Yaskawa INFORM job: X2_DOD_HARDOX_1(90,180).JBI

/JOB
//NAME X2_DOD_HARDOX_1(90,180)
//POS
///NPOS 279,279,279,21,0,0
///TOOL 0
///POSTYPE PULSE
///PULSE
C00000=3109,-122452,-100913,-73,83322,449
C00001=-118807,-122452,-100913,-73,83322,449
C00002=-118807,-122452,-100913,-73,83322,449
C00003=-118807,-122452,-100911,-58,83321,449
C00004=-118807,-121735,-99413,-58,82766,449
C00005=-118807,-121842,-99633,-58,82848,449
C00006=-118839,-119744,-98985,-56,83526,438
C00007=-118804,-122923,-101491,-58,83435,450
C00008=-97639,-115747,-96446,15703,79249,7339
C00009=-97639,-115388,-95597,15719,78924,7296
C00010=-97639,-114939,-94559,15740,78531,7244
C00011=-97639,-115025,-94759,15735,78607,7253
C00012=-98061,-112826,-94039,15753,79350,7198
C00013=-97812,-116320,-99930,15652,81066,7508
C00014=-101587,-63576,-81599,5795,100855,28886
C00015=-101047,-68280,-81443,-762,96025,52675
C00016=-101825,-68101,-80196,-684,95342,52421
C00017=-101825,-68359,-78475,-683,94153,52425
C00018=-101825,-68340,-78625,-683,94255,52425
C00019=-102365,-71446,-80148,-632,93594,52249
C00020=-101826,-68339,-78622,-682,94255,52423
C00021=-102743,-68014,-78460,-592,94316,52120
C00022=-104230,-67130,-78018,-446,94488,51627
C00023=-101826,-68180,-79726,-683,95016,52419
C00024=-105406,-85017,-88644,8711,87087,51760
C00025=-104819,-84637,-86896,8622,86156,51894
C00026=-104819,-84584,-85262,8627,85189,51829
C00027=-104821,-84590,-85434,8628,85291,51834
C00028=-104466,-81413,-84026,8564,86011,52005
C00029=-122297,-70560,-77685,25207,96114,48988
C00030=-122297,-70602,-76512,25163,95437,48844
C00031=-120462,-72211,-77291,25034,94575,49337
C00032=-120807,-72109,-79837,25145,96151,49547
C00033=-93546,-62658,-75100,22039,90269,58200
C00034=-94184,-63290,-73954,22130,89476,57830
C00035=-94067,-63307,-72915,22106,88843,57754
C00036=-94003,-63340,-73099,22003,88907,57787
C00037=-94409,-63618,-73243,22068,88963,57653
C00038=-94117,-63207,-75013,22033,90096,57964
C00039=-99361,-30382,-55480,23023,95964,57224
C00040=-99566,-28855,-54147,23052,95988,57159
C00041=-99566,-29275,-52787,22997,95015,56970
C00042=-99566,-29231,-52941,23002,95123,56991
C00043=-99913,-29435,-53082,23054,95198,56882
C00044=-99765,-28813,-54689,23103,96366,57161
C00045=-70126,-14814,-46677,22990,86577,66649
C00046=-69225,-6747,-37988,28306,84286,67688
C00047=-68210,-7965,-38259,28007,83556,67874
C00048=-68210,-8415,-36953,28052,82637,67651
C00049=-68211,-8369,-37103,28046,82745,67677
C00050=-67132,-7971,-36789,27709,82413,67989
C00051=-68211,-8369,-37103,28046,82745,67677
C00052=-69273,3622,-28812,29896,91299,69888
C00053=-69171,1587,-30541,29875,91281,69920
C00054=-67356,-7788,-38801,27721,83669,68208
C00055=-69304,23814,-19677,20373,105408,54389
C00056=-63772,25809,-17813,13128,104960,54938
C00057=-63772,25417,-17229,13089,104414,54876
C00058=-63772,25480,-17328,13095,104505,54886
C00059=-64757,25100,-17697,13206,104683,54580
C00060=-63772,25480,-17328,13095,104505,54886
C00061=-68307,7319,-30798,19970,94187,53100
C00062=-68472,9999,-28438,20005,94151,53039
C00063=-64638,26032,-18396,13259,105551,54716
C00064=-73474,52417,-1620,14466,110043,52326
C00065=-77083,27840,-18357,21376,94830,50068
C00066=-77083,27429,-17836,21353,94333,49979
C00067=-77083,27542,-17981,21360,94470,50004
C00068=-77263,29809,-15685,21397,94280,49912
C00069=-77083,27542,-17981,21360,94470,50004
C00070=-83249,15329,-22913,33380,85893,48144
C00071=-82325,15284,-22953,33088,85562,48389
C00072=-77119,30179,-17426,21415,95423,50164
C00073=-76952,50122,-2257,13631,106723,63183
C00074=-76686,48992,-1778,13529,105834,63166
C00075=-76686,48070,-780,13449,104775,63046
C00076=-76686,48153,-875,13455,104873,63057
C00077=-76611,45681,-3555,13472,105231,63123
C00078=-76686,48153,-875,13455,104873,63057
C00079=-77765,47797,-1260,13598,105089,62727
C00080=-77503,48179,-2005,13615,105687,62882
C00081=-102232,64721,13378,16026,108849,55032
C00082=-108949,82207,34418,16047,106253,52367
C00083=-109653,82825,36624,15990,105380,52004
C00084=-109653,82216,37670,15908,104457,51880
C00085=-109653,82279,37553,15917,104559,51893
C00086=-109965,79801,34505,15982,105197,51872
C00087=-109653,82279,37553,15917,104559,51893
C00088=-109989,64914,17803,16949,99513,51403
C00089=-109412,64226,17005,16864,99534,51598
C00090=-110036,80923,34280,16050,105899,51944
C00091=-104345,57087,4731,-4349,89209,83366
C00092=-104496,43008,-4738,-4784,85361,83353
C00093=-104479,42314,-3820,-4795,84443,83394
C00094=-104496,42365,-3916,-4789,84527,83385
C00095=-104255,44770,-1355,-4879,84201,83473
C00096=-104496,42365,-3916,-4789,84527,83385
C00097=-105699,43472,-2745,-4351,84311,83020
C00098=-104155,44462,-3948,-4908,85640,83449
C00099=-104173,44480,-3904,-4901,85622,83444
C00100=-106809,29779,-23791,-3960,104541,82225
C00101=-101987,32580,-18779,-13564,104520,81725
C00102=-101987,31981,-18214,-13517,103880,81798
C00103=-101987,32158,-18384,-13531,104070,81776
C00104=-101545,36557,-13887,-13574,103641,81966
C00105=-101545,36395,-13728,-13561,103461,81987
C00106=-101706,33738,-16315,-13551,103657,81914
C00107=-101764,35134,-16470,-13596,104438,81806
C00108=-104548,23177,-32201,15979,107404,88348
C00109=-105455,19857,-30331,15882,104803,87705
C00110=-105493,19341,-29883,15843,104288,87624
C00111=-105493,19514,-30048,15860,104471,87649
C00112=-105050,22772,-26945,15761,104169,87752
C00113=-105050,22547,-26726,15741,103926,87719
C00114=-105181,21576,-27656,15770,104020,87688
C00115=-105214,23260,-28464,15890,105337,87854
C00116=-132284,21592,-30078,20050,110667,79822
C00117=-127713,47562,-3500,19091,106863,80708
C00118=-127298,48428,-1312,18938,105922,80691
C00119=-127298,47930,-750,18875,105351,80598
C00120=-127298,48117,-965,18899,105568,80634
C00121=-126552,50894,2078,18759,104988,80792
C00122=-126552,50661,2355,18730,104712,80748
C00123=-126852,49777,1385,18779,104913,80679
C00124=-126833,51121,1366,18850,105576,80792
C00125=-130599,55255,6018,19225,105667,79530
C00126=-130503,55108,6106,19201,105525,79539
C00127=-130503,54617,6701,19135,104939,79443
C00128=-130503,54765,6517,19154,105119,79472
C00129=-129703,58202,10396,18998,104360,79621
C00130=-129703,58014,10641,18975,104124,79585
C00131=-129980,56421,8841,19034,104460,79543
C00132=-129931,58896,8732,19166,105718,79766
C00133=-131687,18895,-22844,22845,77130,75091
C00134=-123291,20715,-19983,19085,74393,77453
C00135=-123291,20226,-19115,19152,73648,77333
C00136=-123291,20408,-19449,19125,73931,77379
C00137=-123978,17743,-21949,19433,74239,77195
C00138=-123978,17498,-21504,19467,73861,77134
C00139=-123624,18839,-20254,19309,73708,77231
C00140=-123896,19533,-21399,19345,74771,77313
C00141=-129275,29738,-11535,21888,75238,75561
C00142=-129239,30151,-9876,21947,74475,75432
C00143=-129239,29906,-9384,21989,74076,75357
C00144=-129239,29966,-9509,21979,74176,75376
C00145=-128682,29827,-9665,21723,74091,75555
C00146=-129188,29970,-9523,21952,74204,75400
C00147=-129412,25077,-15126,21963,75128,75497
C00148=-127801,23871,-15548,21269,74401,75919
C00149=-127478,25278,-14188,21132,74217,75998
C00150=-127515,25076,-16775,21017,75619,76237
C00151=-133346,41405,-239,23776,75434,74185
C00152=-133209,40965,432,23780,74810,74105
C00153=-133209,40606,1199,23846,74209,73980
C00154=-133209,40709,971,23826,74386,74016
C00155=-134183,37129,-2750,24201,75064,73812
C00156=-134183,36974,-2419,24229,74805,73759
C00157=-133761,38534,-808,24066,74516,73849
C00158=-133829,37887,-2909,24000,75417,74012
C00159=-156022,88654,55414,33609,74162,65271
C00160=-155367,67510,26868,18073,74568,63363
C00161=-155657,68026,27393,18196,74574,63263
C00162=-155657,67713,28231,18251,73929,63165
C00163=-155657,67848,27854,18227,74216,63209
C00164=-157091,64685,24164,18764,75139,62855
C00165=-157091,64518,24594,18793,74808,62803
C00166=-156451,66014,26335,18558,74384,62959
C00167=-156599,65406,24098,18535,75428,63070
C00168=-129275,29738,-11535,21888,75238,75561
C00169=-129021,46521,3990,22011,82280,76800
C00170=-127853,72870,28739,19070,95872,81441
C00171=-127868,72875,28745,19073,95874,81436
C00172=-128195,57479,12526,19645,90783,80632
C00173=-130174,39740,-1969,24825,82186,79427
C00174=-129425,38207,-3565,24549,82155,79680
C00175=-125055,30126,-11758,22903,81812,81108
C00176=-125820,29533,-14095,23141,83054,81090
C00177=-116935,30569,-15261,-2620,77337,75322
C00178=-116946,32606,-9583,-2640,74890,75373
C00179=-117027,32230,-9962,-2601,74928,75346
C00180=-117027,32230,-9962,-2601,74928,75346
C00181=-116186,24046,-15173,-4825,69577,75450
C00182=-116977,23560,-15650,-4179,69663,75252
C00183=-117705,24065,-15165,-3796,69592,75013
C00184=-121349,29184,-10162,-1867,69024,73811
C00185=-155953,64784,27397,14502,67420,61519
C00186=-160308,74014,38140,24557,70405,61761
C00187=-162428,80563,46699,30040,71499,61878
C00188=-162835,78141,41049,29865,73587,62284
C00189=-131165,66178,18557,19074,103796,79028
C00190=-132263,70632,26138,21339,107315,79548
C00191=-130805,66688,21488,21399,107742,80153
C00192=-126998,57798,11204,21464,108466,81651
C00193=-126971,60939,9833,21835,110752,82102
C00194=-128691,16256,-41784,23758,119313,83319
C00195=-126023,-4907,-54781,25051,118959,68774
C00196=-124897,-8515,-53636,24373,116335,68560
C00197=-119086,-23897,-66107,13265,108526,66827
C00198=-120519,-17402,-59352,23947,114251,69687
C00199=-120519,-17402,-59352,23947,114251,69687
C00200=-122564,-44453,-75136,25957,97391,66445
C00201=-123228,-71474,-85542,26631,77979,61978
C00202=-105873,-76739,-89965,2224,72297,65038
C00203=-111330,-72335,-87900,4522,73506,63229
C00204=-111330,-72335,-87900,4522,73506,63229
C00205=-112163,-45580,-78612,3641,93445,63594
C00206=-119086,-23897,-66107,13265,108526,66827
C00207=-125757,-8552,-54820,24574,117205,68447
C00208=-88641,48412,-4226,20715,106428,79236
C00209=-87799,48144,-1656,20397,104625,79199
C00210=-87620,46255,-1934,20290,103831,79122
C00211=-86307,38945,-9666,20202,104482,79674
C00212=-86372,39978,-10015,20293,105198,79777
C00213=-77383,-1492,-44705,4977,83394,77592
C00214=-77548,-1237,-43087,5052,82544,77506
C00215=-83219,23182,-25333,15019,98405,78867
C00216=-80942,13133,-33032,25463,110902,83847
C00217=-81045,14451,-33580,25670,111852,84035
C00218=-73165,-12601,-57571,12637,98383,82001
C00219=-73127,-13258,-56291,12584,97280,81900
C00220=-74782,-8289,-52590,17954,103500,83219
C00221=-74719,-7609,-53088,18001,104113,83334
C00222=-82838,36617,-17283,19543,106393,81060
C00223=-68187,-8044,-38286,28001,83527,67876
C00224=-68187,-8044,-38286,28001,83527,67876
C00225=-67058,-9477,-38022,27689,82372,68007
C00226=-68116,3817,-27265,27987,82912,67789
C00227=-68116,3817,-27265,27987,82912,67789
C00228=-64919,-4904,-34321,21162,76650,66545
C00229=-61528,17256,-21731,13706,92976,69906
C00230=-58415,32145,-10038,7508,102141,70514
C00231=-57465,27559,-14703,8015,104960,71103
C00232=-57465,27559,-14703,8015,104960,71103
C00233=-65198,47488,8134,19223,111073,70945
C00234=-67034,-9554,-38047,27682,82343,68009
C00235=-67251,-9396,-39953,27695,83527,68213
C00236=-83600,19181,-26002,32561,94222,65167
C00237=-77066,27753,-18406,21371,94813,50070
C00238=-76689,29778,-15601,21234,94082,50062
C00239=-76186,35433,-13032,12668,99412,49208
C00240=-76186,35433,-13032,12668,99412,49208
C00241=-74826,30522,-18009,8636,97794,54751
C00242=-79416,42076,-6372,17402,103035,66342
C00243=-86419,39929,-2219,28404,103150,66219
C00244=-84052,39875,-2276,28113,102413,66901
C00245=-84052,39875,-2276,28113,102413,66901
C00246=-81568,19785,-21142,23805,91116,64901
C00247=-82431,9786,-27697,23195,82999,70057
C00248=-82776,9522,-31565,23250,85160,70361
C00249=-89191,6029,-42138,6806,101823,66252
C00250=-95828,93776,43903,513,93919,62536
C00251=-104499,43028,-4714,-4783,85356,83352
C00252=-108433,63055,13709,2825,95010,83470
C00253=-107826,61367,13148,420,94873,83225
C00254=-107008,65665,17554,6129,98722,84709
C00255=-107008,65665,17554,6129,98722,84709
C00256=-106682,56060,7916,7154,93832,84823
C00257=-104948,47222,-158,3217,88060,84363
C00258=-103642,41840,-4077,-3525,83464,83442
C00259=-105882,43444,-2375,-2683,83163,82753
C00260=-105882,43444,-2375,-2683,83163,82753
C00261=-104950,42848,-3229,-5574,83910,82481
C00262=-107826,61367,13148,420,94873,83225
C00263=-106192,65684,14431,-2737,97774,82157
C00264=-82945,4708,-44686,-381,111426,77490
C00265=-79819,-2415,-47658,-697,109614,78498
C00266=-78726,-4935,-47947,-802,108508,78855
C00267=-78978,-4815,-47850,-776,108508,78773
C00268=-82498,-4521,-47863,-435,108644,77640
C00269=-91525,7946,-35181,-15697,111008,71310
C00270=-91286,10128,-36695,-15968,113029,71106
C00271=-98325,-60487,-84418,-569,84750,74718
C00272=-131349,-72907,-81893,29779,75628,65053
C00273=-129293,-70616,-79214,29166,74512,65558
C00274=-88918,-58369,-72899,11987,66692,79059
C00275=-87177,-56818,-72056,11108,66724,79688
C00276=-87910,-58429,-75945,11347,68359,79585
C00277=-85222,-130765,-111241,11638,52830,79008
C00278=3322,-122452,-100913,-73,83322,449
BC00000=198923,666220,911653
BC00001=316579,666220,219283
BC00002=307984,758478,148723
BC00003=307985,760782,131305
BC00004=307985,760782,131305
BC00005=307985,760782,131305
BC00006=307985,760782,131305
BC00007=307985,760782,131305
BC00008=307985,760782,131305
BC00009=307985,760782,131305
BC00010=307985,760782,131305
BC00011=307985,760782,131305
BC00012=307985,760782,131305
BC00013=307985,760782,131305
BC00014=307985,760782,131305
BC00015=307985,760782,131305
BC00016=307985,760782,131305
BC00017=307985,760782,131305
BC00018=307985,760782,131305
BC00019=307985,760782,131305
BC00020=307985,760782,131305
BC00021=307985,760782,131305
BC00022=307985,760782,131305
BC00023=307985,760782,131305
BC00024=307985,760782,131305
BC00025=307985,760782,131305
BC00026=307985,760782,131305
BC00027=307985,760782,131305
BC00028=307985,760782,131305
BC00029=307985,760782,131305
BC00030=307985,760782,131305
BC00031=307985,760782,131305
BC00032=307985,760782,131305
BC00033=307986,760782,131302
BC00034=307986,760782,131302
BC00035=307986,760782,131302
BC00036=307986,760782,131302
BC00037=307986,760782,131302
BC00038=307986,760782,131302
BC00039=307986,760782,131302
BC00040=307986,760782,131302
BC00041=307986,760782,131302
BC00042=307986,760782,131302
BC00043=307986,760782,131302
BC00044=307986,760782,131302
BC00045=258907,777593,97712
BC00046=258907,777593,97712
BC00047=258907,777593,97712
BC00048=258907,777593,97712
BC00049=258907,777592,97711
BC00050=258907,777592,97711
BC00051=258907,777592,97711
BC00052=258907,777592,97711
BC00053=258907,777592,97711
BC00054=258907,777592,97711
BC00055=274910,772479,88149
BC00056=274910,772479,88149
BC00057=274910,772479,88149
BC00058=274910,772479,88149
BC00059=274910,772479,88149
BC00060=274910,772479,88149
BC00061=274910,772479,88149
BC00062=274910,772479,88149
BC00063=274910,772479,88149
BC00064=280793,772479,47450
BC00065=280793,772479,47450
BC00066=280793,772479,47450
BC00067=280793,772479,47450
BC00068=280793,772479,47450
BC00069=280793,772479,47450
BC00070=280793,772479,47450
BC00071=280793,772479,47450
BC00072=280793,772479,47450
BC00073=280793,772479,47450
BC00074=280793,772479,47450
BC00075=280793,772479,47450
BC00076=280793,772479,47450
BC00077=280793,772479,47450
BC00078=280793,772479,47450
BC00079=280793,772479,47450
BC00080=280793,772479,47450
BC00081=311515,772478,37762
BC00082=328438,772478,37762
BC00083=328438,772478,37762
BC00084=328438,772478,37762
BC00085=328438,772478,37762
BC00086=328438,772478,37762
BC00087=328438,772478,37762
BC00088=328438,772478,37762
BC00089=328438,772478,37762
BC00090=328438,772478,37762
BC00091=328438,772478,37762
BC00092=328438,772478,37762
BC00093=328438,772478,37762
BC00094=328438,772478,37762
BC00095=328438,772478,37762
BC00096=328438,772478,37762
BC00097=328438,772478,37762
BC00098=328438,772478,37762
BC00099=308564,725534,37762
BC00100=308564,725534,37762
BC00101=308564,725534,37762
BC00102=308564,725534,37762
BC00103=308564,725534,37762
BC00104=308564,725534,37762
BC00105=308564,725534,37762
BC00106=308564,725534,37762
BC00107=308564,725534,37762
BC00108=308564,725534,37762
BC00109=308564,725534,37762
BC00110=308564,725534,37762
BC00111=308564,725534,37762
BC00112=308564,725534,37762
BC00113=308564,725534,37762
BC00114=308564,725534,37762
BC00115=308564,725534,37762
BC00116=308564,725534,37762
BC00117=308564,725534,37762
BC00118=308564,725534,37762
BC00119=308564,725534,37762
BC00120=308564,725534,37762
BC00121=308564,725534,37762
BC00122=308564,725534,37762
BC00123=308564,725534,37762
BC00124=308564,725534,37762
BC00125=308564,725534,37762
BC00126=308564,725534,37762
BC00127=308564,725534,37762
BC00128=308564,725534,37762
BC00129=308564,725534,37762
BC00130=308564,725534,37762
BC00131=308564,725534,37762
BC00132=308564,725534,37762
BC00133=308564,725534,37762
BC00134=308564,725534,37762
BC00135=308564,725534,37762
BC00136=308564,725534,37762
BC00137=308564,725534,37762
BC00138=308564,725534,37762
BC00139=308564,725534,37762
BC00140=308564,725534,37762
BC00141=308564,725534,37762
BC00142=308564,725534,37762
BC00143=308564,725534,37762
BC00144=308564,725534,37762
BC00145=308564,725534,37762
BC00146=308564,725534,37762
BC00147=308564,725534,37762
BC00148=308564,725534,37762
BC00149=308564,725534,37762
BC00150=308564,725534,37762
BC00151=308564,725534,37761
BC00152=308564,725534,37761
BC00153=308564,725534,37761
BC00154=308564,725534,37761
BC00155=308564,725534,37761
BC00156=308564,725534,37761
BC00157=308564,725534,37761
BC00158=308564,725534,37761
BC00159=362000,725534,37761
BC00160=362000,752970,37761
BC00161=362000,752970,37761
BC00162=362000,752970,37761
BC00163=362000,752970,37761
BC00164=362000,752970,37761
BC00165=362000,752970,37761
BC00166=362000,752970,37761
BC00167=362000,752970,37761
BC00168=308564,725534,37762
BC00169=308564,725534,37762
BC00170=308564,725534,37762
BC00171=308564,725534,37762
BC00172=308564,725534,37762
BC00173=308564,725534,37762
BC00174=308564,725534,37762
BC00175=308564,725534,37762
BC00176=308564,725534,37762
BC00177=308564,725534,37762
BC00178=308564,725534,37762
BC00179=308564,725534,37762
BC00180=308564,725534,37762
BC00181=308564,725534,37762
BC00182=308564,725534,37762
BC00183=308564,725534,37762
BC00184=308564,725534,37762
BC00185=362000,752970,37761
BC00186=362000,752970,37761
BC00187=362000,752970,37761
BC00188=362000,752970,37761
BC00189=308564,725534,37762
BC00190=308564,725534,37762
BC00191=308564,725534,37762
BC00192=308564,725534,37762
BC00193=308564,725534,37762
BC00194=308564,725534,37762
BC00195=308564,725534,37762
BC00196=308564,725534,37762
BC00197=308564,725534,37762
BC00198=308564,725534,37762
BC00199=308564,725534,37762
BC00200=308564,725534,37762
BC00201=308564,725534,37762
BC00202=308564,725534,37762
BC00203=308564,725534,37762
BC00204=308564,725534,37762
BC00205=308564,725534,37762
BC00206=308564,725534,37762
BC00207=308564,725534,37762
BC00208=255253,725534,37762
BC00209=255253,725534,37762
BC00210=255253,725534,37762
BC00211=255253,725534,37762
BC00212=255253,725534,37762
BC00213=255253,725534,37762
BC00214=255254,725534,37762
BC00215=255253,725534,37762
BC00216=255253,725534,37762
BC00217=255253,725534,37762
BC00218=255253,725534,37762
BC00219=255253,725534,37762
BC00220=255253,725534,37762
BC00221=255253,725534,37762
BC00222=255253,725534,37762
BC00223=258907,777593,97712
BC00224=258907,777593,97712
BC00225=258907,777593,97712
BC00226=259033,777461,97560
BC00227=259033,777461,97560
BC00228=259039,777455,97553
BC00229=259039,777455,97553
BC00230=259100,772345,97480
BC00231=259100,773616,97479
BC00232=259100,773616,97479
BC00233=261144,764069,97479
BC00234=258907,777593,97712
BC00235=258907,777593,97712
BC00236=281642,777593,57012
BC00237=280793,772479,47450
BC00238=280794,772478,47449
BC00239=280809,772452,47444
BC00240=280809,772452,47444
BC00241=280809,772452,47444
BC00242=280808,772453,47444
BC00243=293831,772390,68911
BC00244=293831,772390,68911
BC00245=293831,772390,68911
BC00246=293831,772390,68911
BC00247=293831,772390,68911
BC00248=293831,772390,68911
BC00249=293831,772390,68911
BC00250=293831,746596,7862
BC00251=328438,772478,37762
BC00252=328438,772478,37762
BC00253=328438,772478,37762
BC00254=328370,772478,37776
BC00255=328370,772478,37776
BC00256=328370,772478,37776
BC00257=328370,772478,37776
BC00258=328280,772478,37857
BC00259=328280,772478,37857
BC00260=328280,772478,37857
BC00261=328280,772478,37857
BC00262=328438,772478,37762
BC00263=328280,772478,37857
BC00264=293831,772391,68907
BC00265=293831,772391,68906
BC00266=293831,772391,68906
BC00267=293831,772391,68906
BC00268=293831,772391,68906
BC00269=293831,772391,68906
BC00270=293831,772391,68906
BC00271=274540,694640,68906
BC00272=274540,694640,68906
BC00273=274540,694640,68906
BC00274=274540,694640,68906
BC00275=274540,694640,68906
BC00276=274540,694640,68906
BC00277=274540,694640,68906
BC00278=87761,666220,1075229
EC00000=798156,1112951
EC00001=798156,1112951
EC00002=798156,1112951
EC00003=798155,1112950
EC00004=798155,1112950
EC00005=798155,1112950
EC00006=798155,1112950
EC00007=798155,1112950
EC00008=798155,1112950
EC00009=798155,1112950
EC00010=798155,1112950
EC00011=798155,1112950
EC00012=798155,1112950
EC00013=798155,1112950
EC00014=798155,1112950
EC00015=798155,1112950
EC00016=798155,1112950
EC00017=798155,1112950
EC00018=798155,1112950
EC00019=798155,1112950
EC00020=798147,1112941
EC00021=798147,1112941
EC00022=798147,1112941
EC00023=798147,1112941
EC00024=798155,1112950
EC00025=798155,1112950
EC00026=798155,1112950
EC00027=798155,1112950
EC00028=798155,1112950
EC00029=798155,1112950
EC00030=798155,1112950
EC00031=798155,1112950
EC00032=798155,1112950
EC00033=798155,1112949
EC00034=798155,1112949
EC00035=798155,1112949
EC00036=798155,1112949
EC00037=798155,1112949
EC00038=798155,1112949
EC00039=798155,1112949
EC00040=798155,1112949
EC00041=798155,1112949
EC00042=798155,1112949
EC00043=798155,1112949
EC00044=798155,1112949
EC00045=798154,1112948
EC00046=798154,1112948
EC00047=798154,1112948
EC00048=798154,1112948
EC00049=798153,1112947
EC00050=798153,1112947
EC00051=798153,1112947
EC00052=798153,1112947
EC00053=798153,1112947
EC00054=798153,1112947
EC00055=798153,1112947
EC00056=798153,1112947
EC00057=798153,1112947
EC00058=798153,1112947
EC00059=798153,1112947
EC00060=798153,1112947
EC00061=798153,1112947
EC00062=798153,1112947
EC00063=798153,1112947
EC00064=798153,1112947
EC00065=798153,1112947
EC00066=798153,1112947
EC00067=798153,1112947
EC00068=798153,1112947
EC00069=798153,1112947
EC00070=798153,1112947
EC00071=798153,1112947
EC00072=798153,1112947
EC00073=798153,1112947
EC00074=798153,1112947
EC00075=798153,1112947
EC00076=798153,1112947
EC00077=798153,1112947
EC00078=798153,1112947
EC00079=798153,1112947
EC00080=798153,1112947
EC00081=798153,1112946
EC00082=798153,1112946
EC00083=798153,1112946
EC00084=798153,1112946
EC00085=798153,1112946
EC00086=798153,1112946
EC00087=798153,1112946
EC00088=798153,1112946
EC00089=798153,1112946
EC00090=798153,1112946
EC00091=798153,1112946
EC00092=798153,1112946
EC00093=798153,1112946
EC00094=798153,1112946
EC00095=798153,1112946
EC00096=798153,1112946
EC00097=798153,1112946
EC00098=798153,1112946
EC00099=798153,1112946
EC00100=798153,1112946
EC00101=798153,1112946
EC00102=798153,1112946
EC00103=798153,1112946
EC00104=798153,1112946
EC00105=798153,1112946
EC00106=798153,1112946
EC00107=798153,1112946
EC00108=798153,1112946
EC00109=798153,1112946
EC00110=798153,1112946
EC00111=798153,1112946
EC00112=798153,1112946
EC00113=798153,1112946
EC00114=798153,1112946
EC00115=798153,1112946
EC00116=798153,1112946
EC00117=798153,1112946
EC00118=798153,1112946
EC00119=798153,1112946
EC00120=798153,1112946
EC00121=798153,1112946
EC00122=798153,1112946
EC00123=798153,1112946
EC00124=798153,1112946
EC00125=798153,1112946
EC00126=798153,1112946
EC00127=798153,1112946
EC00128=798153,1112946
EC00129=798153,1112946
EC00130=798153,1112946
EC00131=798153,1112946
EC00132=798153,1112946
EC00133=798153,1112946
EC00134=798153,1112946
EC00135=798153,1112946
EC00136=798153,1112946
EC00137=798153,1112946
EC00138=798153,1112946
EC00139=798153,1112946
EC00140=798153,1112946
EC00141=798153,1112946
EC00142=798153,1112946
EC00143=798153,1112946
EC00144=798153,1112946
EC00145=798153,1112946
EC00146=798153,1112946
EC00147=798153,1112946
EC00148=798153,1112946
EC00149=798153,1112946
EC00150=798153,1112946
EC00151=798152,1112944
EC00152=798152,1112944
EC00153=798152,1112944
EC00154=798152,1112944
EC00155=798152,1112944
EC00156=798152,1112944
EC00157=798152,1112944
EC00158=798152,1112944
EC00159=798152,1112944
EC00160=798152,1112944
EC00161=798152,1112944
EC00162=798152,1112944
EC00163=798152,1112944
EC00164=798152,1112944
EC00165=798152,1112944
EC00166=798152,1112944
EC00167=798152,1112944
EC00168=798153,1112946
EC00169=798153,1112946
EC00170=798153,1112946
EC00171=798153,1112946
EC00172=798153,1112946
EC00173=798153,1112946
EC00174=798153,1112946
EC00175=798153,1112946
EC00176=798153,1112946
EC00177=798153,1112946
EC00178=798153,1112946
EC00179=798153,1112946
EC00180=798153,1112946
EC00181=798153,1112946
EC00182=798153,1112946
EC00183=798153,1112946
EC00184=798153,1112946
EC00185=798152,1112944
EC00186=798152,1112944
EC00187=798152,1112944
EC00188=798152,1112944
EC00189=798153,1112946
EC00190=798153,1112946
EC00191=798153,1112946
EC00192=798153,1112946
EC00193=798153,1112946
EC00194=798153,1112946
EC00195=798153,1112946
EC00196=798153,1112946
EC00197=798153,1112946
EC00198=798153,1112946
EC00199=798153,1112946
EC00200=798153,1112946
EC00201=798153,1112946
EC00202=798153,1112946
EC00203=798153,1112946
EC00204=798153,1112946
EC00205=798153,1112946
EC00206=798153,1112946
EC00207=798153,1112946
EC00208=798153,1112946
EC00209=798153,1112946
EC00210=798153,1112946
EC00211=798153,1112946
EC00212=798153,1112946
EC00213=798153,1112946
EC00214=798152,1112945
EC00215=798153,1112946
EC00216=798153,1112946
EC00217=798153,1112946
EC00218=798153,1112946
EC00219=798153,1112946
EC00220=798153,1112946
EC00221=798153,1112946
EC00222=798153,1112946
EC00223=798154,1112948
EC00224=798154,1112948
EC00225=798154,1112948
EC00226=798154,1112948
EC00227=798154,1112948
EC00228=798154,1112948
EC00229=798154,1112948
EC00230=798154,1112948
EC00231=798153,1112947
EC00232=798153,1112947
EC00233=798153,1112947
EC00234=798154,1112948
EC00235=798154,1112948
EC00236=798154,1112948
EC00237=798153,1112947
EC00238=798153,1112946
EC00239=798153,1112946
EC00240=798153,1112946
EC00241=798153,1112946
EC00242=798152,1112944
EC00243=798152,1112944
EC00244=798152,1112944
EC00245=798152,1112944
EC00246=798152,1112944
EC00247=798152,1112944
EC00248=798152,1112944
EC00249=798152,1112944
EC00250=798152,1112944
EC00251=798153,1112946
EC00252=798153,1112946
EC00253=798153,1112946
EC00254=798153,1112946
EC00255=798153,1112946
EC00256=798153,1112946
EC00257=798153,1112946
EC00258=798153,1112946
EC00259=798153,1112946
EC00260=798153,1112946
EC00261=798153,1112946
EC00262=798153,1112946
EC00263=798153,1112946
EC00264=798151,1112943
EC00265=798151,1112942
EC00266=798151,1112942
EC00267=798151,1112942
EC00268=798151,1112942
EC00269=798151,1112942
EC00270=798151,1112942
EC00271=798151,1112942
EC00272=798151,1112942
EC00273=798151,1112942
EC00274=798151,1112942
EC00275=798151,1112942
EC00276=798151,1112942
EC00277=798151,1112942
EC00278=798156,1112951
///POSTYPE BASE
///RECTAN
///RCONF 0,0,0,0,0,0,0,0,0,0,0,0,0,0,0,0,0,0,0,0,0,0,0,0
P00006=0.222,-3.123,-1.508,0.0000,0.0000,0.0000
P00021=-0.225,-6.128,-0.405,0.0000,0.0000,0.0000
P00022=0.222,-3.123,-1.508,0.0000,0.0000,0.0000
P00023=0.143,-0.036,0.682,0.0000,0.0000,0.0000
P00024=0.145,-0.552,1.326,0.0000,0.0000,0.0000
P00025=-2.003,0.006,0.728,0.0000,0.0000,0.0000
P00026=0.562,-0.002,-0.337,0.0000,0.0000,0.0000
P00027=-0.746,0.015,-9.096,0.0000,0.0000,0.0000
P00028=-2.237,-0.018,-7.702,0.0000,0.0000,0.0000
P00029=-2.156,-0.086,-4.681,0.0000,0.0000,0.0000
P00030=5.926,-4.294,-1.390,0.0000,0.0000,0.0000
P00031=1.853,-0.001,-1.549,0.0000,0.0000,0.0000
P00032=1.957,0.503,-7.217,0.0000,0.0000,0.0000
///RCONF 0,0,0,0,1,0,0,0,0,0,0,0,0,0,0,0,0,0,0,0,0,0,0,0
P00033=-0.123,0.612,-5.012,0.0000,0.0000,0.0000
///RCONF 0,0,0,0,0,0,0,0,0,0,0,0,0,0,0,0,0,0,0,0,0,0,0,0
P00034=-0.304,0.773,-2.693,0.0000,0.0000,0.0000
P00035=2.817,0.591,-1.622,0.0000,0.0000,0.0000
P00036=-1.108,-0.829,1.850,0.0000,0.0000,0.0000
P00037=0.023,0.937,-2.677,0.0000,0.0000,0.0000
P00038=0.158,-1.133,-1.952,0.0000,0.0000,0.0000
P00039=0.012,-3.081,-0.106,0.0000,0.0000,0.0000
P00040=-0.030,9.648,2.467,0.0000,0.0000,0.0000
//INST
///DATE 2025/03/13 13:01
///ATTR SC,RW
///GROUP1 RB1,BS1
///GROUP2 ST1
NOP
MOVJ C00000 BC00000 VJ=100.00  +MOVJ EC00000 VJ=100.00
MOVJ C00001 BC00001 VJ=100.00  +MOVJ EC00001 VJ=100.00
MOVL C00002 BC00002 V=1000.0  +MOVJ EC00002 VJ=30.00
SFTOF3D
SMOVL C00003 BC00003 V=166.7  +MOVJ EC00003
SREFP 3 C00004 BC00004  +REFP EC00004
CALL JOB:SEARCH-R1-S13D
SET P021 P006
SFTON3D P021
SMOVL C00005 BC00005 V=166.7  +MOVJ EC00005
SREFP 3 C00006 BC00006  +REFP EC00006
CALL JOB:SEARCH-R1-S13D
SET P021 P006
SFTON3D P021
SMOVL C00007 BC00007 V=166.7  +MOVJ EC00007
SFTOF3D
MOVL C00008 BC00008 V=1000.0  +MOVJ EC00008 VJ=30.00
SMOVL C00009 BC00009 V=166.7  +MOVJ EC00009
SREFP 3 C00010 BC00010  +REFP EC00010
CALL JOB:SEARCH-R1-S13D
SET P022 P006
SFTON3D P022
SMOVL C00011 BC00011 V=166.7  +MOVJ EC00011
SREFP 3 C00012 BC00012  +REFP EC00012
CALL JOB:SEARCH-R1-S13D
SET P022 P006
SFTON3D P022
SMOVL C00013 BC00013 V=166.7  +MOVJ EC00013
MOVJ C00014 BC00014 VJ=30.00  +MOVJ EC00014 VJ=30.00
MOVJ C00015 BC00015 VJ=30.00  +MOVJ EC00015 VJ=30.00
SMOVL C00016 BC00016 V=166.7  +MOVJ EC00016
SREFP 3 C00017 BC00017  +REFP EC00017
CALL JOB:SEARCH-R1-S13D
SET P023 P006
SFTON3D P023
SMOVL C00018 BC00018 V=166.7  +MOVJ EC00018
SREFP 3 C00019 BC00019  +REFP EC00019
CALL JOB:SEARCH-R1-S13D
SET P023 P006
SFTON3D P023
SMOVL C00020 BC00020 V=166.7  +MOVJ EC00020
SMOVL C00021 BC00021 V=166.7  +MOVJ EC00021
SREFP 3 C00022 BC00022  +REFP EC00022
CALL JOB:SEARCH-R1-S13D
SET P023 P006
SFTON3D P023
SMOVL C00023 BC00023 V=166.7  +MOVJ EC00023
MOVJ C00024 BC00024 VJ=30.00  +MOVJ EC00024 VJ=30.00
SMOVL C00025 BC00025 V=166.7  +MOVJ EC00025
SREFP 3 C00026 BC00026  +REFP EC00026
CALL JOB:SEARCH-R1-S13D
SET P024 P006
SFTON3D P024
SMOVL C00027 BC00027 V=166.7  +MOVJ EC00027
SREFP 3 C00028 BC00028  +REFP EC00028
CALL JOB:SEARCH-R1-S13D
SET P024 P006
SFTON3D P024
SMOVL C00029 BC00029 V=333.3  +MOVJ EC00029
SMOVL C00030 BC00030 V=166.7  +MOVJ EC00030
SREFP 3 C00031 BC00031  +REFP EC00031
CALL JOB:SEARCH-R1-S13D
SET P024 P006
SFTON3D P024
SMOVL C00032 BC00032 V=333.3  +MOVJ EC00032
SMOVL C00033 BC00033 V=333.3 PL=0  +MOVJ EC00033
SMOVL C00034 BC00034 V=166.7  +MOVJ EC00034
SREFP 3 C00035 BC00035  +REFP EC00035
CALL JOB:SEARCH-R1-S13D
SET P025 P006
SFTON3D P025
SMOVL C00036 BC00036 V=166.7  +MOVJ EC00036
SREFP 3 C00037 BC00037  +REFP EC00037
CALL JOB:SEARCH-R1-S13D
SET P025 P006
SFTON3D P025
SMOVL C00038 BC00038 V=333.3  +MOVJ EC00038
SMOVL C00039 BC00039 V=666.7  +MOVJ EC00039
SMOVL C00040 BC00040 V=166.7  +MOVJ EC00040
SREFP 3 C00041 BC00041  +REFP EC00041
CALL JOB:SEARCH-R1-S13D
SET P026 P006
SFTON3D P026
SMOVL C00042 BC00042 V=166.7  +MOVJ EC00042
SREFP 3 C00043 BC00043  +REFP EC00043
CALL JOB:SEARCH-R1-S13D
SET P026 P006
SFTON3D P026
SMOVL C00044 BC00044 V=333.3  +MOVJ EC00044
MOVL C00045 BC00045 V=666.7  +MOVJ EC00045 VJ=30.00
MOVL C00046 BC00046 V=666.7  +MOVJ EC00046 VJ=30.00
SMOVL C00047 BC00047 V=166.7  +MOVJ EC00047
SREFP 3 C00048 BC00048  +REFP EC00048
CALL JOB:SEARCH-R1-S13D
SET P027 P006
SFTON3D P027
SMOVL C00049 BC00049 V=166.7  +MOVJ EC00049
SREFP 3 C00050 BC00050  +REFP EC00050
CALL JOB:SEARCH-R1-S13D
SET P027 P006
SFTON3D P027
SMOVL C00051 BC00051 V=166.7  +MOVJ EC00051
SMOVL C00052 BC00052 V=166.7  +MOVJ EC00052
SREFP 3 C00053 BC00053  +REFP EC00053
CALL JOB:SEARCH-R1-S13D
SET P027 P006
SFTON3D P027
SMOVL C00054 BC00054 V=333.3  +MOVJ EC00054
MOVL C00055 BC00055 V=666.7  +MOVJ EC00055 VJ=30.00
SMOVL C00056 BC00056 V=166.7  +MOVJ EC00056
SREFP 3 C00057 BC00057  +REFP EC00057
CALL JOB:SEARCH-R1-S13D
SET P028 P006
SFTON3D P028
SMOVL C00058 BC00058 V=166.7  +MOVJ EC00058
SREFP 3 C00059 BC00059  +REFP EC00059
CALL JOB:SEARCH-R1-S13D
SET P028 P006
SFTON3D P028
SMOVL C00060 BC00060 V=166.7  +MOVJ EC00060
SMOVL C00061 BC00061 V=166.7  +MOVJ EC00061
SREFP 3 C00062 BC00062  +REFP EC00062
CALL JOB:SEARCH-R1-S13D
SET P028 P006
SFTON3D P028
SMOVL C00063 BC00063 V=333.3  +MOVJ EC00063
MOVL C00064 BC00064 V=666.7  +MOVJ EC00064 VJ=30.00
SMOVL C00065 BC00065 V=166.7  +MOVJ EC00065
SREFP 3 C00066 BC00066  +REFP EC00066
CALL JOB:SEARCH-R1-S13D
SET P029 P006
SFTON3D P029
SMOVL C00067 BC00067 V=166.7  +MOVJ EC00067
SREFP 3 C00068 BC00068  +REFP EC00068
CALL JOB:SEARCH-R1-S13D
SET P029 P006
SFTON3D P029
SMOVL C00069 BC00069 V=166.7  +MOVJ EC00069
SMOVL C00070 BC00070 V=166.7  +MOVJ EC00070
SREFP 3 C00071 BC00071  +REFP EC00071
CALL JOB:SEARCH-R1-S13D
SET P029 P006
SFTON3D P029
SMOVL C00072 BC00072 V=333.3  +MOVJ EC00072
MOVL C00073 BC00073 V=666.7  +MOVJ EC00073 VJ=30.00
SMOVL C00074 BC00074 V=166.7  +MOVJ EC00074
SREFP 3 C00075 BC00075  +REFP EC00075
CALL JOB:SEARCH-R1-S13D
SET P030 P006
SFTON3D P030
SMOVL C00076 BC00076 V=166.7  +MOVJ EC00076
SREFP 3 C00077 BC00077  +REFP EC00077
CALL JOB:SEARCH-R1-S13D
SET P030 P006
SFTON3D P030
SMOVL C00078 BC00078 V=166.7  +MOVJ EC00078
SREFP 3 C00079 BC00079  +REFP EC00079
CALL JOB:SEARCH-R1-S13D
SET P030 P006
SFTON3D P030
SMOVL C00080 BC00080 V=166.7  +MOVJ EC00080
MOVL C00081 BC00081 V=666.7  +MOVJ EC00081 VJ=30.00
MOVL C00082 BC00082 V=666.7  +MOVJ EC00082 VJ=30.00
SMOVL C00083 BC00083 V=166.7  +MOVJ EC00083
SREFP 3 C00084 BC00084  +REFP EC00084
CALL JOB:SEARCH-R1-S13D
SET P031 P006
SFTON3D P031
SMOVL C00085 BC00085 V=166.7  +MOVJ EC00085
SREFP 3 C00086 BC00086  +REFP EC00086
CALL JOB:SEARCH-R1-S13D
SET P031 P006
SFTON3D P031
SMOVL C00087 BC00087 V=166.7  +MOVJ EC00087
SMOVL C00088 BC00088 V=166.7  +MOVJ EC00088
SREFP 3 C00089 BC00089  +REFP EC00089
CALL JOB:SEARCH-R1-S13D
SET P031 P006
SFTON3D P031
SMOVL C00090 BC00090 V=333.3  +MOVJ EC00090
MOVJ C00091 BC00091 VJ=30.00  +MOVJ EC00091 VJ=30.00
SMOVL C00092 BC00092 V=166.7  +MOVJ EC00092
SREFP 3 C00093 BC00093  +REFP EC00093
CALL JOB:SEARCH-R1-S13D
SET P032 P006
SFTON3D P032
SMOVL C00094 BC00094 V=166.7  +MOVJ EC00094
SREFP 3 C00095 BC00095  +REFP EC00095
CALL JOB:SEARCH-R1-S13D
SET P032 P006
SFTON3D P032
SMOVL C00096 BC00096 V=166.7  +MOVJ EC00096
SREFP 3 C00097 BC00097  +REFP EC00097
CALL JOB:SEARCH-R1-S13D
SET P032 P006
SFTON3D P032
SMOVL C00098 BC00098 V=333.3  +MOVJ EC00098
SFTOF3D
MOVJ C00099 BC00099 VJ=30.00  +MOVJ EC00099 VJ=30.00
MOVJ C00100 BC00100 VJ=30.00  +MOVJ EC00100 VJ=30.00
SMOVL C00101 BC00101 V=166.7  +MOVJ EC00101
SREFP 3 C00102 BC00102  +REFP EC00102
CALL JOB:SEARCH-R1-S13D
SET P033 P006
SFTON3D P033
SMOVL C00103 BC00103 V=166.7  +MOVJ EC00103
SMOVL C00104 BC00104 V=666.7  +MOVJ EC00104
SMOVL C00105 BC00105 V=166.7  +MOVJ EC00105
SREFP 3 C00106 BC00106  +REFP EC00106
CALL JOB:SEARCH-R1-S13D
SET P033 P006
SFTON3D P033
SMOVL C00107 BC00107 V=333.3  +MOVJ EC00107
SFTOF3D
SMOVL C00108 BC00108 V=666.7  +MOVJ EC00108
SMOVL C00109 BC00109 V=166.7  +MOVJ EC00109
SREFP 3 C00110 BC00110  +REFP EC00110
CALL JOB:SEARCH-R1-S13D
SET P034 P006
SFTON3D P034
SMOVL C00111 BC00111 V=166.7  +MOVJ EC00111
SMOVL C00112 BC00112 V=666.7  +MOVJ EC00112
SMOVL C00113 BC00113 V=666.7  +MOVJ EC00113
SREFP 3 C00114 BC00114  +REFP EC00114
CALL JOB:SEARCH-R1-S13D
SET P034 P006
SFTON3D P034
SMOVL C00115 BC00115 V=333.3  +MOVJ EC00115
SFTOF3D
SMOVL C00116 BC00116 V=666.7  +MOVJ EC00116
SMOVL C00117 BC00117 V=666.7  +MOVJ EC00117
SMOVL C00118 BC00118 V=166.7  +MOVJ EC00118
SREFP 3 C00119 BC00119  +REFP EC00119
CALL JOB:SEARCH-R1-S13D
SET P035 P006
SFTON3D P035
SMOVL C00120 BC00120 V=166.7  +MOVJ EC00120
SMOVL C00121 BC00121 V=666.7  +MOVJ EC00121
SMOVL C00122 BC00122 V=666.7  +MOVJ EC00122
SREFP 3 C00123 BC00123  +REFP EC00123
CALL JOB:SEARCH-R1-S13D
SET P035 P006
SFTON3D P035
SMOVL C00124 BC00124 V=333.3  +MOVJ EC00124
SFTOF3D
SMOVL C00125 BC00125 V=666.7  +MOVJ EC00125
SMOVL C00126 BC00126 V=166.7  +MOVJ EC00126
SREFP 3 C00127 BC00127  +REFP EC00127
CALL JOB:SEARCH-R1-S13D
SET P036 P006
SFTON3D P036
SMOVL C00128 BC00128 V=166.7  +MOVJ EC00128
SMOVL C00129 BC00129 V=666.7  +MOVJ EC00129
SMOVL C00130 BC00130 V=666.7  +MOVJ EC00130
SREFP 3 C00131 BC00131  +REFP EC00131
CALL JOB:SEARCH-R1-S13D
SET P036 P006
SFTON3D P036
SMOVL C00132 BC00132 V=333.3  +MOVJ EC00132
SFTOF3D
SMOVL C00133 BC00133 V=666.7  +MOVJ EC00133
SMOVL C00134 BC00134 V=166.7  +MOVJ EC00134
SREFP 3 C00135 BC00135  +REFP EC00135
CALL JOB:SEARCH-R1-S13D
SET P037 P006
SFTON3D P037
SMOVL C00136 BC00136 V=166.7  +MOVJ EC00136
SMOVL C00137 BC00137 V=666.7  +MOVJ EC00137
SMOVL C00138 BC00138 V=666.7  +MOVJ EC00138
SREFP 3 C00139 BC00139  +REFP EC00139
CALL JOB:SEARCH-R1-S13D
SET P037 P006
SFTON3D P037
SMOVL C00140 BC00140 V=333.3  +MOVJ EC00140
SFTOF3D
SMOVL C00141 BC00141 V=666.7  +MOVJ EC00141
SMOVL C00142 BC00142 V=166.7  +MOVJ EC00142
SREFP 3 C00143 BC00143  +REFP EC00143
CALL JOB:SEARCH-R1-S13D
SET P038 P006
SFTON3D P038
SMOVL C00144 BC00144 V=166.7  +MOVJ EC00144
SREFP 3 C00145 BC00145  +REFP EC00145
CALL JOB:SEARCH-R1-S13D
SET P038 P006
SFTON3D P038
SMOVL C00146 BC00146 V=333.3  +MOVJ EC00146
SMOVL C00147 BC00147 V=666.7  +MOVJ EC00147
SMOVL C00148 BC00148 V=666.7  +MOVJ EC00148
SREFP 3 C00149 BC00149  +REFP EC00149
CALL JOB:SEARCH-R1-S13D
SET P038 P006
SFTON3D P038
SMOVL C00150 BC00150 V=333.3  +MOVJ EC00150
SFTOF3D
SMOVL C00151 BC00151 V=666.7  +MOVJ EC00151
SMOVL C00152 BC00152 V=166.7  +MOVJ EC00152
SREFP 3 C00153 BC00153  +REFP EC00153
CALL JOB:SEARCH-R1-S13D
SET P039 P006
SFTON3D P039
SMOVL C00154 BC00154 V=166.7  +MOVJ EC00154
SMOVL C00155 BC00155 V=666.7  +MOVJ EC00155
SMOVL C00156 BC00156 V=666.7  +MOVJ EC00156
SREFP 3 C00157 BC00157  +REFP EC00157
CALL JOB:SEARCH-R1-S13D
SET P039 P006
SFTON3D P039
SMOVL C00158 BC00158 V=333.3  +MOVJ EC00158
SFTOF3D
SMOVL C00159 BC00159 V=666.7  +MOVJ EC00159
SMOVL C00160 BC00160 V=666.7  +MOVJ EC00160
SMOVL C00161 BC00161 V=166.7  +MOVJ EC00161
SREFP 3 C00162 BC00162  +REFP EC00162
CALL JOB:SEARCH-R1-S13D
SET P040 P006
SFTON3D P040
SMOVL C00163 BC00163 V=166.7  +MOVJ EC00163
SMOVL C00164 BC00164 V=666.7  +MOVJ EC00164
SMOVL C00165 BC00165 V=666.7  +MOVJ EC00165
SREFP 3 C00166 BC00166  +REFP EC00166
CALL JOB:SEARCH-R1-S13D
SET P040 P006
SFTON3D P040
SMOVL C00167 BC00167 V=333.3  +MOVJ EC00167
SFTOF3D
SMOVL C00168 BC00168 V=666.7  +MOVJ EC00168
SFTON3D P038
MACRO1 MJ#(0) ARGF9
SMOVL C00169 BC00169 V=150.0 PL=0  +MOVJ EC00169
ARCON
SMOVL C00170 BC00170 V=11.7  +MOVJ EC00170
SMOVC C00171 BC00171 V=13.3  +MOVJ EC00171
SMOVC C00172 BC00172 V=13.3  +MOVJ EC00172
SMOVC C00173 BC00173 V=13.3  +MOVJ EC00173
SMOVL C00174 BC00174 V=11.7  +MOVJ EC00174
SFTON3D P037
SMOVL C00175 BC00175 V=11.7  +MOVJ EC00175
ARCOF
SMOVL C00176 BC00176 V=333.3  +MOVJ EC00176
SSFTOF
SMOVL C00177 BC00177 V=666.7  +MOVJ EC00177
SFTON3D P038
MACRO1 MJ#(0) ARGF9
SMOVL C00178 BC00178 V=150.0 PL=0  +MOVJ EC00178
ARCON
SMOVL C00179 BC00179 V=11.7  +MOVJ EC00179
SMOVC C00180 BC00180 V=13.3  +MOVJ EC00180
SMOVC C00181 BC00181 V=13.3  +MOVJ EC00181
SFTON3D P039
SMOVC C00182 BC00182 V=13.3  +MOVJ EC00182
SMOVL C00183 BC00183 V=11.7  +MOVJ EC00183
MOVL C00184 BC00184 V=11.7  +MOVJ EC00184 VJ=30.00
SFTON3D P040
SMOVL C00185 BC00185 V=11.7  +MOVJ EC00185
MOVL C00186 BC00186 V=11.7  +MOVJ EC00186 VJ=30.00
MOVL C00187 BC00187 V=11.7  +MOVJ EC00187 VJ=30.00
ARCOF
SMOVL C00188 BC00188 V=333.3  +MOVJ EC00188
SSFTOF
MOVL C00189 BC00189 V=666.7  +MOVJ EC00189 VJ=30.00
SFTON3D P036
SMOVL C00190 BC00190 V=150.0 PL=0  +MOVJ EC00190
ARCON
SMOVL C00191 BC00191 V=11.7  +MOVJ EC00191
SFTON3D P035
SMOVL C00192 BC00192 V=11.7  +MOVJ EC00192
ARCOF
MOVL C00193 BC00193 V=333.3  +MOVJ EC00193 VJ=30.00
SFTOF3D
MOVL C00194 BC00194 V=666.7  +MOVJ EC00194 VJ=30.00
MOVL C00195 BC00195 V=666.7  +MOVJ EC00195 VJ=30.00
SFTON3D P023
SMOVL C00196 BC00196 V=666.7  +MOVJ EC00196
SMOVL C00197 BC00197 V=150.0 PL=0  +MOVJ EC00197
ARCON
SFTON3D P024
SMOVL C00198 BC00198 V=11.7  +MOVJ EC00198
SMOVC C00199 BC00199 V=13.3  +MOVJ EC00199
SMOVC C00200 BC00200 V=13.3  +MOVJ EC00200
SMOVC C00201 BC00201 V=13.3  +MOVJ EC00201
SFTON3D P023
SMOVL C00202 BC00202 V=11.7  +MOVJ EC00202
SMOVL C00203 BC00203 V=11.7  +MOVJ EC00203
SMOVC C00204 BC00204 V=13.3  +MOVJ EC00204
SMOVC C00205 BC00205 V=13.3  +MOVJ EC00205
SMOVC C00206 BC00206 V=13.3  +MOVJ EC00206
ARCOF
SMOVL C00207 BC00207 V=333.3  +MOVJ EC00207
SFTOF3D
MOVL C00208 BC00208 V=666.7  +MOVJ EC00208 VJ=30.00
SFTON3D P026
MOVL C00209 BC00209 V=666.7  +MOVJ EC00209 VJ=30.00
SMOVL C00210 BC00210 V=150.0 PL=0  +MOVJ EC00210
ARCON
SWVON WEV#(70)
SMOVL C00211 BC00211 V=6.7  +MOVJ EC00211
ARCOF
SWVOF
SMOVL C00212 BC00212 V=333.3  +MOVJ EC00212
SMOVL C00213 BC00213 V=333.3  +MOVJ EC00213
SMOVL C00214 BC00214 V=150.0 PL=0  +MOVJ EC00214
ARCON
SWVON WEV#(70)
SMOVL C00215 BC00215 V=6.7  +MOVJ EC00215
SFTON3D P025
SMOVL C00216 BC00216 V=6.7  +MOVJ EC00216
ARCOF
SWVOF
SMOVL C00217 BC00217 V=333.3  +MOVJ EC00217
SMOVL C00218 BC00218 V=333.3  +MOVJ EC00218
SMOVL C00219 BC00219 V=150.0 PL=0  +MOVJ EC00219
ARCON
SWVON WEV#(70)
SMOVL C00220 BC00220 V=6.7  +MOVJ EC00220
ARCOF
SWVOF
SMOVL C00221 BC00221 V=333.3  +MOVJ EC00221
SFTOF3D
MOVL C00222 BC00222 V=666.7  +MOVJ EC00222 VJ=30.00
MOVL C00223 BC00223 V=666.7  +MOVJ EC00223 VJ=30.00
SFTON3D P027
SMOVL C00224 BC00224 V=666.7  +MOVJ EC00224
SMOVL C00225 BC00225 V=150.0 PL=0  +MOVJ EC00225
ARCON
SFTON3D P028
SMOVL C00226 BC00226 V=11.7  +MOVJ EC00226
SMOVC C00227 BC00227 V=13.3  +MOVJ EC00227
SMOVC C00228 BC00228 V=13.3  +MOVJ EC00228
SMOVC C00229 BC00229 V=13.3  +MOVJ EC00229
SFTON3D P027
SMOVL C00230 BC00230 V=11.7  +MOVJ EC00230
SMOVL C00231 BC00231 V=11.7  +MOVJ EC00231
SMOVC C00232 BC00232 V=13.3  +MOVJ EC00232
SMOVC C00233 BC00233 V=13.3  +MOVJ EC00233
SMOVC C00234 BC00234 V=13.3  +MOVJ EC00234
ARCOF
SMOVL C00235 BC00235 V=333.3  +MOVJ EC00235
SFTOF3D
MOVL C00236 BC00236 V=666.7  +MOVJ EC00236 VJ=30.00
MOVL C00237 BC00237 V=666.7  +MOVJ EC00237 VJ=30.00
SFTON3D P029
SMOVL C00238 BC00238 V=150.0 PL=0  +MOVJ EC00238
ARCON
SFTON3D P030
SMOVL C00239 BC00239 V=11.7  +MOVJ EC00239
SMOVC C00240 BC00240 V=13.3  +MOVJ EC00240
SMOVC C00241 BC00241 V=13.3  +MOVJ EC00241
SMOVC C00242 BC00242 V=13.3  +MOVJ EC00242
SFTON3D P029
SMOVL C00243 BC00243 V=11.7  +MOVJ EC00243
SMOVL C00244 BC00244 V=11.7  +MOVJ EC00244
SMOVC C00245 BC00245 V=13.3  +MOVJ EC00245
SMOVC C00246 BC00246 V=13.3  +MOVJ EC00246
SMOVC C00247 BC00247 V=13.3  +MOVJ EC00247
ARCOF
SMOVL C00248 BC00248 V=333.3  +MOVJ EC00248
SFTOF3D
MOVL C00249 BC00249 V=666.7  +MOVJ EC00249 VJ=30.00
MOVL C00250 BC00250 V=666.7  +MOVJ EC00250 VJ=30.00
MOVL C00251 BC00251 V=666.7  +MOVJ EC00251 VJ=30.00
SMOVL C00252 BC00252 V=666.7  +MOVJ EC00252
SFTON3D P032
SMOVL C00253 BC00253 V=150.0 PL=0  +MOVJ EC00253
ARCON
SFTON3D P031
SMOVL C00254 BC00254 V=11.7  +MOVJ EC00254
SMOVC C00255 BC00255 V=13.3  +MOVJ EC00255
SMOVC C00256 BC00256 V=13.3  +MOVJ EC00256
SMOVC C00257 BC00257 V=13.3  +MOVJ EC00257
SFTON3D P032
SMOVL C00258 BC00258 V=11.7  +MOVJ EC00258
SMOVL C00259 BC00259 V=11.7  +MOVJ EC00259
SMOVC C00260 BC00260 V=13.3  +MOVJ EC00260
SMOVC C00261 BC00261 V=13.3  +MOVJ EC00261
SMOVC C00262 BC00262 V=13.3  +MOVJ EC00262
ARCOF
SMOVL C00263 BC00263 V=333.3  +MOVJ EC00263
SFTOF3D
MOVL C00264 BC00264 V=666.7  +MOVJ EC00264 VJ=30.00
SFTON3D P034
MOVL C00265 BC00265 V=666.7  +MOVJ EC00265 VJ=30.00
SMOVL C00266 BC00266 V=150.0 PL=0  +MOVJ EC00266
ARCON
SMOVL C00267 BC00267 V=11.7  +MOVJ EC00267
SMOVL C00268 BC00268 V=11.7  +MOVJ EC00268
SFTON3D P033
SMOVL C00269 BC00269 V=11.7  +MOVJ EC00269
ARCOF
SMOVL C00270 BC00270 V=333.3  +MOVJ EC00270
SFTOF3D
MOVL C00271 BC00271 V=666.7  +MOVJ EC00271 VJ=30.00
MOVL C00272 BC00272 V=666.7  +MOVJ EC00272 VJ=30.00
SFTON3D P021
SMOVL C00273 BC00273 V=150.0 PL=0  +MOVJ EC00273
ARCON
SFTON3D P022
SMOVL C00274 BC00274 V=11.7  +MOVJ EC00274
SMOVL C00275 BC00275 V=11.7  +MOVJ EC00275
ARCOF
SMOVL C00276 BC00276 V=333.3  +MOVJ EC00276
SFTOF3D
MOVL C00277 BC00277 V=1000.0  +MOVJ EC00277 VJ=30.00
'
MOVJ C00278 BC00278 VJ=100.00  +MOVJ EC00278 VJ=100.00
END
